{attribute 'qualified_only'}
{attribute 'strict'}
TYPE E_SeqSEW_WithBrake :
(
	INIT := 0,
	STOPPED,
	RELEASE_BRAKE,
	FORWARD,
	BACKWARD,
	STOP,
	APPLY_BRAKE
);
END_TYPE

(* stored: Version 1.1.0.1, ProductVersion 3.1.4024.12
   DUT E_SeqSEW_WithBrake: Id {a7ca8203-6194-4717-902a-e0feabf8114c} *)
